// TIA Portal V17 export
// export: Created 2023-02-14T02:49:36.2635455Z, ExportSetting WithDefaults, DisplayName Totally Integrated Automation Portal, DisplayVersion V17, DisplayName TIA Portal Openness, DisplayVersion V17, DisplayName TIA Portal Teamcenter Gateway, DisplayVersion V17, DisplayName TIA Portal Version Control Interface, DisplayVersion V17, DisplayName SINAMICS Startdrive Advanced, DisplayVersion V17, DisplayName SINAMICS Startdrive G130, G150, S120, S150, SINAMICS MV, S210, DisplayVersion V17, DisplayName SINAMICS Startdrive G110M, G120, G120C, G120D, G120P, G115D, DisplayVersion V17, DisplayName STEP 7 Professional, DisplayVersion V17, DisplayName STEP 7 Safety, DisplayVersion V17, DisplayName WinCC Professional, DisplayVersion V17
DATA_BLOCK "IO_Valve_T04_Chili"   // DB304
VERSION : 0.1
// stored: AutoNumber false, DBAccessibleFromOPCUA true, DBAccessibleFromWebserver true, InstanceOfName IO Valve T04 Chili, InstanceOfType FB
"IO Valve T04 Chili"
   // VAR_INPUT
   //    lock : Bool;
   //    Init : Bool;
   //    testing : Bool;
   //    Reset : Bool;
   // END_VAR
   // VAR
   //    "AV-04.01" { S7_SetPoint := 'True'} : "Valve";
   //    "AV-04.02" { S7_SetPoint := 'True'} : "Valve";
   //    "AV-04.03" { S7_SetPoint := 'True'} : "Valve";
   //    "AV-04.04" { S7_SetPoint := 'True'} : "Valve";
   //    "AV-04.05" { S7_SetPoint := 'True'} : "Valve";
   //    "AV-04.06" { S7_SetPoint := 'True'} : "Valve";
   //    "AV-04.07" { S7_SetPoint := 'True'} : "Valve";
   //    "AV-04.08" { S7_SetPoint := 'True'} : "Valve";
   //    "AV-04.09" { S7_SetPoint := 'True'} : "Valve";
   //    "AV-04.10" { S7_SetPoint := 'True'} : "Valve";
   //    "AV-04.11" { S7_SetPoint := 'True'} : "Valve";
   //    "AV-04.12" { S7_SetPoint := 'True'} : "Valve";
   //    "AV-04.13" { S7_SetPoint := 'True'} : "Valve";
   //    "AV-04.14" { S7_SetPoint := 'True'} : "Valve";
   //    "AV-04.15" { S7_SetPoint := 'True'} : "Valve";
   // END_VAR
BEGIN
END_DATA_BLOCK
